FUNCTION_BLOCK AX_X_TO_BOOL (* Composite FB for convert AX to BOOL *)
  (* Standard: 61499-2; Description: Copyright (c) 2024 HR Agrartechnik GmbH This program and the accompanying materials are made available under the terms of the Eclipse Public License 2.0 which is available at https://www.eclipse.org/legal/epl-2.0/ SPDX-License-Identifier: EPL-2.0 *)
  (* Version 1.0, 2024-04-24, Franz Höpfinger, HR Agrartechnik GmbH *)
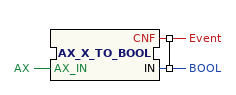
  EVENT_OUTPUT
    CNF WITH IN; (* Confirmation from Adapter *)
  END_EVENT
  VAR_OUTPUT
    IN : BOOL; (* Input data from Adapter *)
  END_VAR
  SOCKETS
    AX_IN : AX; (* Adapter Input *)
  END_SOCKETS
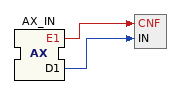
  EVENT_CONNECTIONS
    AX_IN.E1 TO CNF;
  END_CONNECTIONS
  DATA_CONNECTIONS
    AX_IN.D1 TO IN;
  END_CONNECTIONS
END_FUNCTION_BLOCK
